# EPICS substitutions: ipimbIocApp/Db/ioc-xrt-xcsimb1.substitutions
#==============================================================================
#
# Abs:  ipimb Records
#
# Name: ioc-xrt-xcsimb1.substitutions
#
#==============================================================================
#
file ipimb.template
{
	pattern
	{ RECNAME    , BOX      }
	{ HXX:UM6:PIM:01 , HXX-UM6-PIM-01 }
}
